{attribute 'qualified_only'}
{attribute 'strict'}
TYPE E_EventType :
(
	alarm := 0,
	Message := 1
);
END_TYPE

(* stored: Version 1.1.0.1, ProductVersion 3.1.4024.12
   DUT E_EventType: Id {ca16fb1a-de24-4dab-a1d9-edce8e00956d} *)
